TYPE COLLECTION_LENGTH : DINT(0..2147483647); END_TYPE

(* stored: Version 1.1.0.1
   DUT COLLECTION_LENGTH: Id {f9f1e8d3-62bb-482d-a49b-4b08445b7f7d} *)
